(* IEC 61131-3 sources: POMIRTS_lab3/AS/Library_2/ArSafeUDP, 3 files *)

(* ---- ArSafeUDP.typ ---- *)
TYPE

END_TYPE

(* ---- ArSafeUDP.fun ---- *)
{REDUND_CONTEXT} FUNCTION ArSafeUDPEnable  : DINT (*Enable an openSAFETY-over-UDP tunnel.*)
	VAR_INPUT
		DeviceName	: STRING[127]; (*Device name (syntax: SL<a>.SS<b>.IF<c>.ST<d>) of the openSAFETY-over-UDP tunnel.*)
	END_VAR
END_FUNCTION

{REDUND_CONTEXT} FUNCTION ArSafeUDPDisable : DINT (*Disable an openSAFETY-over-UDP tunnel.*)
	VAR_INPUT
		DeviceName	: STRING[127]; (*Device name (syntax: SL<a>.SS<b>.IF<c>.ST<d>) of the openSAFETY-over-UDP tunnel.*)
	END_VAR
END_FUNCTION

{REDUND_CONTEXT} FUNCTION ArSafeUDPSetIP   : DINT (*Change the IP for an openSAFETY-over-UDP tunnel.*)
	VAR_INPUT
		DeviceName	: STRING[127]; (*Device name (syntax: SL<a>.SS<b>.IF<c>.ST<d>) of the openSAFETY-over-UDP tunnel.*)
		IPAddress	: STRING[15]; (*IP address, valid range "1.0.0.1" - "247.255.255.255".*)
	END_VAR
END_FUNCTION

(* ---- ArSafeUDP.var ---- *)
VAR CONSTANT
	arSAFEUDP_ERR_DEV_NOT_FOUND		: DINT := -1070583900;	(*Is returned when no openSAFETY-over-UDP tunnel exists with the given device name.*)
	arSAFEUDP_ERR_TUNNEL_ENABLED	: DINT := -1070583901;	(*Is returned when the openSAFETY-over-UDP tunnel must not be enabled to use this function.*)
	arSAFEUDP_ERR_IP_INVALID		: DINT := -1070583902;	(*Is returned when the given IP is not in the valid range of "1.0.0.1" - "247.255.255.255".*)
	arSAFEUDP_ERR_IP_IN_USE			: DINT := -1070583903;	(*Is returned when the configured IP is already in use by another openSAFETY-over-UDP tunnel.*)
END_VAR
